FUNCTION_BLOCK Conveyor (* Basic Function Block Type *)
  (* Standard: 61499-2 *)
  (* Version 0.0, 2015-03-25, 4DIAC-IDE, 4DIAC-Consortium *)
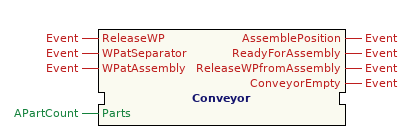
  EVENT_INPUT
    ReleaseWP;
    WPatSeparator;
    WPatAssembly;
  END_EVENT
  EVENT_OUTPUT
    AssemblePosition;
    ReadyForAssembly;
    ReleaseWPfromAssembly;
    ConveyorEmpty;
  END_EVENT
  SOCKETS
    Parts : APartCount;
  END_SOCKETS
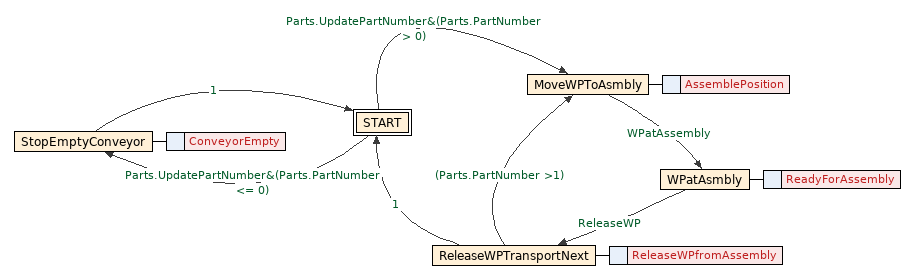
  EC_STATES
    START; (* Initial State *)
    MoveWPToAsmbly : -> AssemblePosition;
    ReleaseWPTransportNext : -> ReleaseWPfromAssembly;
    WPatAsmbly : -> ReadyForAssembly;
    StopEmptyConveyor : -> ConveyorEmpty;
  END_STATES
  EC_TRANSITIONS
    WPatAsmbly TO ReleaseWPTransportNext := ReleaseWP;
    StopEmptyConveyor TO START := 1;
    START TO StopEmptyConveyor := Parts.UpdatePartNumber&(Parts.PartNumber <= 0);
    START TO MoveWPToAsmbly := Parts.UpdatePartNumber&(Parts.PartNumber > 0);
    ReleaseWPTransportNext TO MoveWPToAsmbly := (Parts.PartNumber >1);
    ReleaseWPTransportNext TO START := 1;
    MoveWPToAsmbly TO WPatAsmbly := WPatAssembly;
  END_TRANSITIONS
  SERVICE conveyor_interface/conveyor_implementation (* Basic Function Block Type *)
    SEQUENCE stop_empty_conveyor
      conveyor_interface.Parts.UpdatePartNumber(Parts.PartNumber <= 0) -> conveyor_interface.ConveyorEmpty();
    END_SEQUENCE
    SEQUENCE start_conveyor_0
      conveyor_interface.Parts.UpdatePartNumber(Parts.PartNumber > 0) -> conveyor_interface.AssemblePosition();
      conveyor_interface.WPatAssembly() -> conveyor_interface.ReadyForAssembly();
      conveyor_interface.ReleaseWP() -> conveyor_interface.ReleaseWPfromAssembly();
    END_SEQUENCE
    SEQUENCE start_conveyor_1
      conveyor_interface.Parts.UpdatePartNumber(Parts.PartNumber > 1) -> conveyor_interface.AssemblePosition();
      conveyor_interface.WPatAssembly() -> conveyor_interface.ReadyForAssembly();
      conveyor_interface.ReleaseWP() -> conveyor_interface.ReleaseWPfromAssembly();
    END_SEQUENCE
  END_SERVICE
END_FUNCTION_BLOCK
